// TwinCAT 3 PLC project Plc
// Title: Plc
// Company: TcProberExamples
// ProjectVersion: 0.0.0.1
// ProgramVersion: 3.1.4023.0
// libraries:
//   Tc2_Standard, * (Beckhoff Automation GmbH)
//   Tc2_System, * (Beckhoff Automation GmbH)
//   Tc3_Module, * (Beckhoff Automation GmbH)
// project tree:
//   / fbDrive.TcPOU, fbDriveTest.TcPOU, MAIN_TESTS.TcPOU, PlcTask.TcTTO
// real-time tasks:
//   TASK PlcTask: cycle T#10ms, priority 20, ADS port 350

CONFIGURATION Plc
    RESOURCE PLC ON TwinCAT3
        TASK PlcTask(INTERVAL := T#10ms, PRIORITY := 20);
        PROGRAM MAIN_TESTS WITH PlcTask : MAIN_TESTS;
    END_RESOURCE
END_CONFIGURATION

// ---- MAIN_TESTS.TcPOU
PROGRAM INTERNAL MAIN_TESTS
VAR
	_driveTest : fbDriveTest;
END_VAR

_driveTest();

END_PROGRAM

// ---- fbDriveTest.TcPOU
FUNCTION_BLOCK INTERNAL fbDriveTest
VAR
	_drive : fbDrive;
END_VAR

_drive();

{attribute 'TcRpcEnable'}
METHOD INTERNAL MoveAbsoluteTest : BOOL
VAR_INPUT
	Position : LREAL;
	Speed : LREAL;
	AccDcc : LREAL;
END_VAR
MoveAbsoluteTest := _drive.MoveAbsolute(Position, 
										Speed, 
										AccDcc);
END_METHOD

END_FUNCTION_BLOCK

// ---- fbDrive.TcPOU
FUNCTION_BLOCK fbDrive
VAR	
	_position : LREAL;
	_speed : LREAL;
	_acc_dcc : LREAL;
	
	_targetPosition : LREAL;
	_targetSpeed : LREAL;
	_targetAccDcc : LREAL;
END_VAR
VAR  
	_changextime : LREAL;
END_VAR

_changextime := (_targetSpeed * 0.01);

IF(ABS(_position - _targetPosition) <= _changextime * 2) THEN _position := _targetPosition; RETURN; END_IF;

IF (_position < _targetPosition) THEN _position := _position + _changextime; END_IF;
IF (_position > _targetPosition) THEN _position := _position - _changextime; END_IF;

METHOD MoveAbsolute : BOOL
VAR_INPUT
	Position : LREAL;
	Speed : LREAL;
	AccDcc : LREAL;
END_VAR
_targetPosition := Position;
_targetSpeed := Speed;
_targetAccDcc := AccDcc;

MoveAbsolute := 
     _targetPosition = _position;
END_METHOD

END_FUNCTION_BLOCK
